// TIA Portal V19 export
TYPE "Prod_Part_Done"
// stored: Access Published
   STRUCT
      Done : Bool;   // Target eseguito
      LeadCut : Bool;   // Intestazione
      Weld : Bool;   // La parte ha la saldatura
      Tick_Mark : Bool;   // E' stato eseguito il Marchio identificazione spessore
      Trace_Mark : Bool;   // E' stato eseguito il Marchio identificazione tracciabilità
      P_ID : DInt;   // ID pezzo assegnato al pezzo eseguito
      O_ID : DInt;   // ID di produzione a cui appartiene la parte da fare
      Part_LenMeas : Real;   // Lunghezza della parte misurata
   END_STRUCT;
END_TYPE
